(*
	Clamp the input value within the range of 0 to 1
*)
FUNCTION F_Clamp01 : REAL
VAR_INPUT
	fValue : REAL;
END_VAR

F_Clamp01:= LIMIT(0, fValue, 1);

END_FUNCTION

(* stored: Version 1.1.0.1, ProductVersion 3.1.4024.12
   POU F_Clamp01: Id {8b7c9793-6c86-01cf-298d-98158576c883}, SpecialFunc None *)
